Universal Robots URScript: spheremod.script

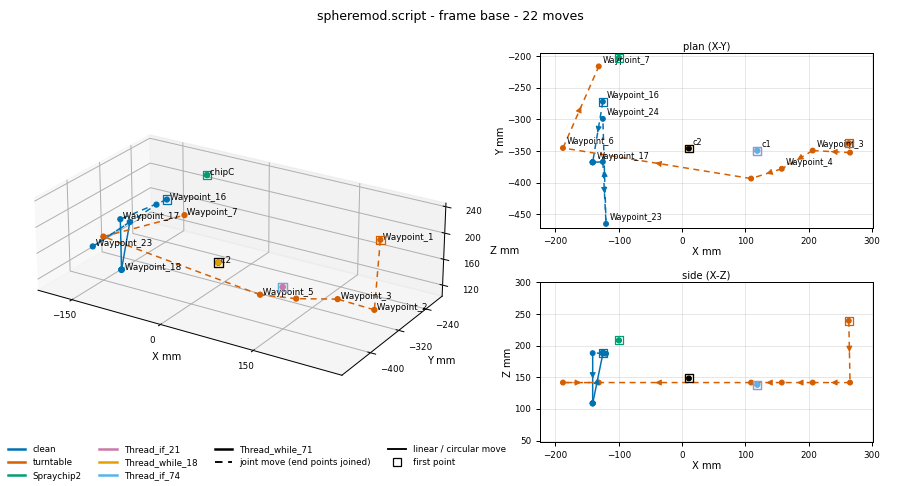
[picture p0: tool path of spheremod.script in frame base, 22 of 62 moves have a stored position in this frame; points joined in program order, loops and branches not executed]
def spheremod():
  global _hidden_verificationVariable=0
  step_count_fb48d3ff_0c9f_4d99_a765_ea41926c28d5 = 0.0
  thread Step_Counter_Thread_a9617a2c_6c0b_4ca4_aaba_c79477845290():
    while (True):
      step_count_fb48d3ff_0c9f_4d99_a765_ea41926c28d5 = step_count_fb48d3ff_0c9f_4d99_a765_ea41926c28d5 + 1.0
      sync()
    end
  end
  run Step_Counter_Thread_a9617a2c_6c0b_4ca4_aaba_c79477845290()
  set_standard_analog_input_domain(0, 1)
  set_standard_analog_input_domain(1, 1)
  set_tool_analog_input_domain(0, 1)
  set_tool_analog_input_domain(1, 1)
  set_analog_outputdomain(0, 0)
  set_analog_outputdomain(1, 0)
  set_input_actions_to_default()
  set_tool_communication(False, 115200, 0, 1, 1.5, 3.5)
  set_tool_output_mode(0)
  set_tool_digital_output_mode(0, 1)
  set_tool_digital_output_mode(1, 1)
  set_tool_voltage(0)
  set_safety_mode_transition_hardness(1)
  set_gravity([0.0, 0.0, 9.82])
  set_target_payload(0.530000, [0.009000, -0.039000, 0.092000], [0.000534, 0.000534, 0.000534, 0.000000, 0.000000, 0.000000])
  set_tcp(p[0.0,0.0,0.11,0.0,0.0,0.0])
  global Al_plate=p[0.12405209206180495,-0.2666666051843552,0.020008101224669964,-9.276623980477388E-5,1.8107917580596192E-5,3.1233857134705927]
  global Frame2x2=p[0.18266245434305164,-0.34273121659514855,0.026002571110600767,-2.225423529876215E-4,3.0110667546023537E-4,3.1233976058306383]
  global Plane_1=p[0.0,0.0,0.0,0.0,0.0,0.0]
  global URlogoTutorial=p[-0.08178353973148575,-0.3363174165299142,0.04788621506469384,-3.9746155723688456E-5,-3.4682148779121894E-5,-1.5668291789091222]
  global carousel=p[0.13865255139760183,-0.25132593351268107,0.051531504137083003,-4.453572132438073E-5,-1.3071222590669835E-4,-3.1349676625391965]
  global carouselrod=p[0.2020731702281844,-0.34951442511341274,0.1947611446273096,3.139766958234101,-0.10689428010274801,-1.1796370330365635E-5]
  global paper=p[-0.09670794781244417,-0.3283412964648025,0.027665994240809913,-3.2057893450593004E-5,2.867088716161181E-5,-1.6085327915291054]
  global rod=p[0.13368013097420872,-0.41123185103490206,0.09926814901395645,2.2214229924093103,-2.2214158162465862,-2.9165882738638143E-5]
  global timer_1=0
  global c1_p=p[.118888830935, -.349388142069, .138324188628, -3.141139658809, .028493427521, .002872972354]
  global c1_q=[-0.8784921805011194, -1.7871462307372035, -1.5894867181777954, -1.3364218038371583, 1.5709693431854248, 3.850743532180786]
  global c2_p=p[.010821857253, -.346022311091, .148298540443, -3.141186124538, .028346003463, .002753345138]
  global c2_q=[-1.1497486273394983, -1.679014345208639, -1.6702346801757812, -1.3633616727641602, 1.5705503225326538, 3.57938551902771]
  global Waypoint_16_p=p[-.125097928533, -.271984222044, .188211676824, -3.139810722578, .105446315311, .000070958927]
  global Waypoint_16_q=[-1.5480602423297327, -1.4491210740855713, -1.7099264860153198, -1.552596167927124, 1.5715936422348022, 3.23006010055542]
  global Waypoint_17_p=p[-.141183217597, -.367684006591, .188213447751, 3.139821760490, -.105397104768, -.000067867997]
  global Waypoint_17_q=[-1.597567383443014, -1.8740092716612757, -1.241610050201416, -1.5960084400572718, 1.5719740390777588, 3.1803600788116455]
  global Waypoint_18_p=p[-.141178244459, -.367687282910, .108904454765, 3.139816402425, -.105408093734, -.000060814483]
  global Waypoint_18_q=[-1.5975983778582972, -1.9245020351805628, -1.550661325454712, -1.2364590925029297, 1.5723340511322021, 3.1807193756103516]
  global Waypoint_19_p=p[-.141189357305, -.367687267469, .108915260822, 3.121780755938, .351957921543, -.000099281586]
  global Waypoint_19_q=[-1.5976179281817835, -1.9244748554625453, -1.550661325454712, -1.2364507478526612, 1.572314977645874, 2.889045000076294]
  global Waypoint_20_p=p[-.141176698746, -.367682773595, .108907204798, -3.111042719163, .436975672702, .000063164110]
  global Waypoint_20_q=[-1.5975945631610315, -1.9244939289488734, -1.5506495237350464, -1.2365017098239441, 1.5723340511322021, 3.3926987648010254]
  global Waypoint_21_p=p[-.141174078526, -.367696805030, .108909057026, 3.139786221315, -.105395786134, -.000060564502]
  global Waypoint_21_q=[-1.597586456929342, -1.9245058498778285, -1.5506460666656494, -1.2364399594119568, 1.5723340511322021, 3.1807241439819336]
  global Waypoint_22_p=p[-.125093999497, -.367099400456, .187371407622, 3.139783011421, -.105392168035, -.000053869150]
  global Waypoint_22_q=[-1.5538747946368616, -1.846323629418844, -1.2822730541229248, -1.5829936466612757, 1.5719654560089111, 3.224064588546753]
  global Waypoint_23_p=p[-.120064390322, -.465070651334, .187365924664, 2.700279766902, -.088400420341, .019763045538]
  global Waypoint_23_q=[-1.5412524382220667, -1.9475652180113734, -1.406833291053772, -0.9173591893962403, 1.5603561401367188, 3.2332537174224854]
  global Waypoint_24_p=p[-.125099110421, -.299097154487, .189878767902, 3.139750209928, -.105401717856, -.000111797080]
  global Waypoint_24_q=[-1.550074879323141, -1.5617311683348198, -1.5979981422424316, -1.5518303674510499, 1.5716702938079834, 3.2279696464538574]
  global Waypoint_1_p=p[.263501689877, -.337317763427, .239349489480, 3.139797243720, -.105347053477, -.000037720516]
  global Waypoint_1_q=[-0.5959728399859827, -2.1057659588255824, -0.6533136367797852, -1.9525557957091273, 1.5718059539794922, 4.181682586669922]
  global Waypoint_2_p=p[.265438435610, -.352444474661, .141740907029, 3.139726376264, -.105360108121, -.000022031768]
  global Waypoint_2_q=[-0.6231134573565882, -2.1016999683775843, -1.126999020576477, -1.4828875821879883, 1.5722739696502686, 4.154912948608398]
  global Waypoint_3_p=p[.206441973084, -.349241721273, .141737893294, 3.139734184252, -.105329347268, -.000022485776]
  global Waypoint_3_q=[-0.7073677221881312, -1.9410401783385218, -1.3681066036224365, -1.4024366003325959, 1.5721865892410278, 4.070710182189941]
  global Waypoint_4_p=p[.157616611756, -.378012026932, .141738203587, 3.139764187573, -.105376653239, -.000076760662]
  global Waypoint_4_q=[-0.8494070211993616, -1.9579774341978968, -1.3439116477966309, -1.409730003481247, 1.5722019672393799, 3.928692579269409]
  global Waypoint_5_p=p[.109134761588, -.393436595889, .141742225598, 3.139732501163, -.105376381431, -.000050533951]
  global Waypoint_5_q=[-0.972816292439596, -1.9523960552611292, -1.3519116640090942, -1.4072665137103577, 1.5721949338912964, 3.805286407470703]
  global Waypoint_6_p=p[-.188131250090, -.345166366147, .141750553976, 3.139727051239, -.105353578209, -.000024875816]
  global Waypoint_6_q=[-1.7293437162982386, -1.8864180050291957, -1.4439769983291626, -1.381135032778122, 1.572224736213684, 3.0487747192382812]
  global Waypoint_7_p=p[-.131564048097, -.216205376465, .141741700579, 3.139714533984, -.105382776464, -.000044168049]
  global Waypoint_7_q=[-1.572542969380514, -1.2417927545360108, -2.0833356380462646, -1.3863917154124756, 1.571577787399292, 3.2058310508728027]
  global chipC_p=p[-.099703384862, -.202952364142, .208439850600, 3.139657619359, -.105437397760, -.000145108772]
  global chipC_q=[-1.4082325140582483, -1.0998719197562714, -1.8470008373260498, -1.7646123371519984, 1.5710017681121826, 3.3699307441711426]
  global Waypoint_15_p=p[-.099704296715, -.202951379992, .208432580258, 3.139670120847, -.105426183766, -.000160358536]
  global Waypoint_15_q=[-1.4082286993609827, -1.099871740942337, -1.8470300436019897, -1.764597078362936, 1.5709946155548096, 3.369927167892456]
  global timer_1_is_counting=False
  thread Timer_Thread():
    while (True):
      if (timer_1_is_counting):
        timer_1 = timer_1 + get_steptime()
      end
      sync()
    end
  end
  run Timer_Thread()
  def CircleAllangles():
    $ 181 "CircleAllangles" "noBreak"
    $ 182 "p0≔p[c[0]+r,c[1],c[2],c[3],c[4],c[5]-1.5*A]"
    global p0=p[c[0]+r,c[1],c[2],c[3],c[4],c[5]-1.5*A]
    $ 183 "p45≔p[c[0]+0.71*r,c[1]+0.71*r,c[2],c[3]-A/1.1,c[4],c[5]-A/1.1]"
    global p45=p[c[0]+0.71*r,c[1]+0.71*r,c[2],c[3]-A/1.1,c[4],c[5]-A/1.1]
    $ 184 "p90≔p[c[0],c[1]+r,c[2],c[3]-A,c[4],c[5]]"
    global p90=p[c[0],c[1]+r,c[2],c[3]-A,c[4],c[5]]
    $ 185 "p135≔p[c[0]-0.71*r,c[1]+0.71*r,c[2],c[3]-A/1.1,c[4],c[5]+A/1.1]"
    global p135=p[c[0]-0.71*r,c[1]+0.71*r,c[2],c[3]-A/1.1,c[4],c[5]+A/1.1]
    $ 186 "p180≔p[c[0]-r,c[1],c[2],c[3],c[4],c[5]+1.5*A]"
    global p180=p[c[0]-r,c[1],c[2],c[3],c[4],c[5]+1.5*A]
    $ 187 "p225≔p[c[0]-0.71*r,c[1]-0.71*r,c[2],c[3]+A/1.1,c[4],c[5]+A/1.1]"
    global p225=p[c[0]-0.71*r,c[1]-0.71*r,c[2],c[3]+A/1.1,c[4],c[5]+A/1.1]
    $ 188 "p270≔p[c[0],c[1]-r,c[2],c[3]+A,c[4],c[5]]"
    global p270=p[c[0],c[1]-r,c[2],c[3]+A,c[4],c[5]]
    $ 189 "p315≔p[c[0]+0.71*r,c[1]-0.71*r,c[2],c[3]+A/1.1,c[4],c[5]-A/1.1]"
    global p315=p[c[0]+0.71*r,c[1]-0.71*r,c[2],c[3]+A/1.1,c[4],c[5]-A/1.1]
    $ 190 "Set atomization=On"
    set_standard_digital_out(1, True)
    $ 191 "Set triggersolenoid=On"
    set_standard_digital_out(0, True)
    $ 192 "MoveL"
    $ 193 "p0" "breakAfter"
    set_tcp(p[0.0,0.0,0.11,0.0,0.0,0.0])
    movel(p0, a=1.3, v=0.35, r=0.005)
    $ 195 "p45" "breakAfter"
    set_tcp(p[0.0,0.0,0.11,0.0,0.0,0.0])
    movel(p45, a=1.3, v=0.35, r=0.005)
    $ 197 "p90" "breakAfter"
    set_tcp(p[0.0,0.0,0.11,0.0,0.0,0.0])
    movel(p90, a=1.3, v=0.35, r=0.005)
    $ 199 "p135" "breakAfter"
    set_tcp(p[0.0,0.0,0.11,0.0,0.0,0.0])
    movel(p135, a=1.3, v=0.35, r=0.005)
    $ 201 "p180" "breakAfter"
    set_tcp(p[0.0,0.0,0.11,0.0,0.0,0.0])
    movel(p180, a=1.3, v=0.35, r=0.005)
    $ 206 "p225" "breakAfter"
    set_tcp(p[0.0,0.0,0.11,0.0,0.0,0.0])
    movel(p225, a=1.3, v=0.35, r=0.005)
    $ 208 "p270" "breakAfter"
    set_tcp(p[0.0,0.0,0.11,0.0,0.0,0.0])
    movel(p270, a=1.3, v=0.35, r=0.005)
    $ 210 "p315" "breakAfter"
    set_tcp(p[0.0,0.0,0.11,0.0,0.0,0.0])
    movel(p315, a=1.3, v=0.35, r=0.005)
    $ 212 "p0" "breakAfter"
    set_tcp(p[0.0,0.0,0.11,0.0,0.0,0.0])
    movel(p0, a=1.3, v=0.35, r=0.005)
    $ 214 "p45" "breakAfter"
    set_tcp(p[0.0,0.0,0.11,0.0,0.0,0.0])
    movel(p45, a=1.3, v=0.35, r=0.005)
    $ 219 "p90" "breakAfter"
    set_tcp(p[0.0,0.0,0.11,0.0,0.0,0.0])
    movel(p90, a=1.3, v=0.35, r=0.005)
    $ 226 "Set atomization=Off"
    set_standard_digital_out(1, False)
    $ 227 "Set triggersolenoid=Off"
    set_standard_digital_out(0, False)
  end
  def clean():
    $ 228 "clean" "noBreak"
    $ 229 "MoveJ"
    $ 230 "Waypoint_16" "breakAfter"
    movej(get_inverse_kin(Waypoint_16_p, qnear=Waypoint_16_q), a=1.3962634015954636, v=1.0471975511965976)
    $ 231 "Waypoint_17" "breakAfter"
    movej(get_inverse_kin(Waypoint_17_p, qnear=Waypoint_17_q), a=1.3962634015954636, v=1.0471975511965976)
    $ 232 "MoveL"
    $ 233 "Waypoint_18" "breakAfter"
    movel(Waypoint_18_p, a=1.2, v=0.05)
    $ 234 "MoveL"
    $ 235 "Waypoint_19" "breakAfter"
    movel(Waypoint_19_p, a=1.2, v=0.05)
    $ 236 "MoveL"
    $ 237 "Waypoint_20" "breakAfter"
    movel(Waypoint_20_p, a=1.2, v=0.05)
    $ 238 "MoveL"
    $ 239 "Waypoint_21" "breakAfter"
    movel(Waypoint_21_p, a=1.2, v=0.05)
    $ 240 "MoveL"
    $ 241 "Waypoint_22" "breakAfter"
    movel(Waypoint_22_p, a=1.2, v=0.25)
    $ 242 "MoveJ"
    $ 243 "Waypoint_23" "breakAfter"
    movej(get_inverse_kin(Waypoint_23_p, qnear=Waypoint_23_q), a=1.3962634015954636, v=1.0471975511965976)
    $ 244 "Set atomization=On"
    set_standard_digital_out(1, True)
    $ 245 "Set triggersolenoid=On"
    set_standard_digital_out(0, True)
    $ 246 "Wait: 0.2"
    sleep(0.2)
    $ 247 "Set atomization=Off"
    set_standard_digital_out(1, False)
    $ 248 "Set triggersolenoid=Off"
    set_standard_digital_out(0, False)
    $ 249 "MoveJ"
    $ 250 "Waypoint_24" "breakAfter"
    movej(get_inverse_kin(Waypoint_24_p, qnear=Waypoint_24_q), a=1.3962634015954636, v=1.0471975511965976)
  end
  def turntable():
    $ 251 "turntable" "noBreak"
    $ 252 "MoveJ"
    $ 253 "Waypoint_1" "breakAfter"
    set_tcp(p[0.0,0.0,0.11,0.0,0.0,0.0])
    movej(get_inverse_kin(pose_trans(carouselrod, pose_trans(p[-.225374943892, -.334963115589, .194760490875, -3.139766958133, .106894280099, .000011796372], Waypoint_1_p)), qnear=Waypoint_1_q), a=1.3962634015954636, v=0.5235987755982988, r=0.02)
    $ 254 "Waypoint_2" "breakAfter"
    set_tcp(p[0.0,0.0,0.11,0.0,0.0,0.0])
    movej(get_inverse_kin(pose_trans(carouselrod, pose_trans(p[-.225374943892, -.334963115589, .194760490875, -3.139766958133, .106894280099, .000011796372], Waypoint_2_p)), qnear=Waypoint_2_q), a=1.3962634015954636, v=0.5235987755982988, r=0.02)
    $ 255 "Waypoint_3" "breakAfter"
    set_tcp(p[0.0,0.0,0.11,0.0,0.0,0.0])
    movej(get_inverse_kin(pose_trans(carouselrod, pose_trans(p[-.225374943892, -.334963115589, .194760490875, -3.139766958133, .106894280099, .000011796372], Waypoint_3_p)), qnear=Waypoint_3_q), a=1.3962634015954636, v=0.5235987755982988, r=0.02)
    $ 256 "Waypoint_4" "breakAfter"
    set_tcp(p[0.0,0.0,0.11,0.0,0.0,0.0])
    movej(get_inverse_kin(pose_trans(carouselrod, pose_trans(p[-.225374943892, -.334963115589, .194760490875, -3.139766958133, .106894280099, .000011796372], Waypoint_4_p)), qnear=Waypoint_4_q), a=1.3962634015954636, v=0.5235987755982988, r=0.02)
    $ 257 "Waypoint_5" "breakAfter"
    set_tcp(p[0.0,0.0,0.11,0.0,0.0,0.0])
    movej(get_inverse_kin(pose_trans(carouselrod, pose_trans(p[-.225374943892, -.334963115589, .194760490875, -3.139766958133, .106894280099, .000011796372], Waypoint_5_p)), qnear=Waypoint_5_q), a=1.3962634015954636, v=0.5235987755982988, r=0.02)
    $ 258 "MoveJ"
    $ 259 "Waypoint_6" "breakAfter"
    movej(get_inverse_kin(pose_trans(carouselrod, pose_trans(p[-.225374943892, -.334963115589, .194760490875, -3.139766958133, .106894280099, .000011796372], Waypoint_6_p)), qnear=Waypoint_6_q), a=1.3962634015954636, v=0.3141592653589793)
    $ 260 "Wait: 1.0"
    sleep(1.0)
    $ 261 "MoveJ"
    $ 262 "Waypoint_7" "breakAfter"
    movej(get_inverse_kin(pose_trans(carouselrod, pose_trans(p[-.225374943892, -.334963115589, .194760490875, -3.139766958133, .106894280099, .000011796372], Waypoint_7_p)), qnear=Waypoint_7_q), a=1.3962634015954636, v=1.0471975511965976, r=0.02)
  end
  def Spraychip2():
    $ 263 "Spraychip2" "noBreak"
    $ 264 "MoveJ"
    $ 265 "chipC" "breakAfter"
    movej(get_inverse_kin(chipC_p, qnear=chipC_q), a=1.3962634015954636, v=1.0471975511965976)
    $ 266 "c≔chipC"
    global c=chipC_p
    $ 267 "rc≔27/1000"
    global rc=27/1000
    $ 268 "p0≔p[c[0]+rc,c[1],c[2],c[3],c[4],c[5]-1.5*0]"
    global p0=p[c[0]+rc,c[1],c[2],c[3],c[4],c[5]-1.5*0]
    $ 269 "p45≔p[c[0]+0.71*rc,c[1]+0.71*rc,c[2],c[3]-0/1.1,c[4],c[5]-0/1.1]"
    global p45=p[c[0]+0.71*rc,c[1]+0.71*rc,c[2],c[3]-0/1.1,c[4],c[5]-0/1.1]
    $ 270 "p90≔p[c[0],c[1]+rc,c[2],c[3]-0,c[4],c[5]]"
    global p90=p[c[0],c[1]+rc,c[2],c[3]-0,c[4],c[5]]
    $ 271 "p135≔p[c[0]-0.71*rc,c[1]+0.71*rc,c[2],c[3]-0/1.1,c[4],c[5]+0/1.1]"
    global p135=p[c[0]-0.71*rc,c[1]+0.71*rc,c[2],c[3]-0/1.1,c[4],c[5]+0/1.1]
    $ 272 "p180≔p[c[0]-rc,c[1],c[2],c[3],c[4],c[5]+1.5*0]"
    global p180=p[c[0]-rc,c[1],c[2],c[3],c[4],c[5]+1.5*0]
    $ 273 "p225≔p[c[0]-0.71*rc,c[1]-0.71*rc,c[2],c[3]+0/1.1,c[4],c[5]+0/1.1]"
    global p225=p[c[0]-0.71*rc,c[1]-0.71*rc,c[2],c[3]+0/1.1,c[4],c[5]+0/1.1]
    $ 274 "p270≔p[c[0],c[1]-rc,c[2],c[3]+0,c[4],c[5]]"
    global p270=p[c[0],c[1]-rc,c[2],c[3]+0,c[4],c[5]]
    $ 275 "p315≔p[c[0]+0.71*rc,c[1]-0.71*rc,c[2],c[3]+0/1.1,c[4],c[5]-0/1.1]"
    global p315=p[c[0]+0.71*rc,c[1]-0.71*rc,c[2],c[3]+0/1.1,c[4],c[5]-0/1.1]
    $ 276 "Set atomization=On"
    set_standard_digital_out(1, True)
    $ 277 "Set triggersolenoid=On"
    set_standard_digital_out(0, True)
    $ 278 "MoveL"
    $ 279 "p0" "breakAfter"
    set_tcp(p[0.0,0.0,0.11,0.0,0.0,0.0])
    movel(p0, a=1.3, v=0.085, r=0.01)
    $ 280 "p45" "breakAfter"
    set_tcp(p[0.0,0.0,0.11,0.0,0.0,0.0])
    movel(p45, a=1.3, v=0.085, r=0.01)
    $ 281 "p90" "breakAfter"
    set_tcp(p[0.0,0.0,0.11,0.0,0.0,0.0])
    movel(p90, a=1.3, v=0.085, r=0.01)
    $ 282 "p135" "breakAfter"
    set_tcp(p[0.0,0.0,0.11,0.0,0.0,0.0])
    movel(p135, a=1.3, v=0.085, r=0.01)
    $ 283 "p180" "breakAfter"
    set_tcp(p[0.0,0.0,0.11,0.0,0.0,0.0])
    movel(p180, a=1.3, v=0.085, r=0.01)
    $ 284 "Set triggersolenoid=Off"
    set_standard_digital_out(0, False)
    $ 285 "Wait: 0.1"
    sleep(0.1)
    $ 286 "Set triggersolenoid=On"
    set_standard_digital_out(0, True)
    $ 287 "p225" "breakAfter"
    set_tcp(p[0.0,0.0,0.11,0.0,0.0,0.0])
    movel(p225, a=1.3, v=0.085, r=0.01)
    $ 288 "p270" "breakAfter"
    set_tcp(p[0.0,0.0,0.11,0.0,0.0,0.0])
    movel(p270, a=1.3, v=0.085, r=0.01)
    $ 289 "p315" "breakAfter"
    set_tcp(p[0.0,0.0,0.11,0.0,0.0,0.0])
    movel(p315, a=1.3, v=0.085, r=0.01)
    $ 290 "p0" "breakAfter"
    set_tcp(p[0.0,0.0,0.11,0.0,0.0,0.0])
    movel(p0, a=1.3, v=0.085, r=0.01)
    $ 291 "p45" "breakAfter"
    set_tcp(p[0.0,0.0,0.11,0.0,0.0,0.0])
    movel(p45, a=1.3, v=0.085, r=0.01)
    $ 292 "Set triggersolenoid=Off"
    set_standard_digital_out(0, False)
    $ 293 "Wait: 0.1"
    sleep(0.1)
    $ 294 "Set triggersolenoid=On"
    set_standard_digital_out(0, True)
    $ 295 "p90" "breakAfter"
    set_tcp(p[0.0,0.0,0.11,0.0,0.0,0.0])
    movel(p90, a=1.3, v=0.085, r=0.01)
    $ 296 "p135" "breakAfter"
    set_tcp(p[0.0,0.0,0.11,0.0,0.0,0.0])
    movel(p135, a=1.3, v=0.085, r=0.01)
    $ 297 "p180" "breakAfter"
    set_tcp(p[0.0,0.0,0.11,0.0,0.0,0.0])
    movel(p180, a=1.3, v=0.085, r=0.01)
    $ 298 "p225" "breakAfter"
    set_tcp(p[0.0,0.0,0.11,0.0,0.0,0.0])
    movel(p225, a=1.3, v=0.085, r=0.01)
    $ 299 "p270" "breakAfter"
    set_tcp(p[0.0,0.0,0.11,0.0,0.0,0.0])
    movel(p270, a=1.3, v=0.085, r=0.01)
    $ 300 "p315" "breakAfter"
    set_tcp(p[0.0,0.0,0.11,0.0,0.0,0.0])
    movel(p315, a=1.3, v=0.085, r=0.01)
    $ 301 "p0" "breakAfter"
    set_tcp(p[0.0,0.0,0.11,0.0,0.0,0.0])
    movel(p0, a=1.3, v=0.085, r=0.01)
    $ 302 "MoveJ"
    $ 303 "Waypoint_15" "breakAfter"
    movej(get_inverse_kin(Waypoint_15_p, qnear=Waypoint_15_q), a=1.3962634015954636, v=1.0471975511965976)
    $ 304 "Wait: 0.2"
    sleep(0.2)
    $ 305 "Set atomization=Off"
    set_standard_digital_out(1, False)
    $ 306 "Set triggersolenoid=Off"
    set_standard_digital_out(0, False)
  end
  while (True):
    $ 2 "Robot Program"
    $ 3 "'Program to be used for part #124517-035 sphere mod'"
    # 'Program to be used for part #124517-035 sphere mod'
    $ 4 "'Program rev ___: mm/dd/yy note'"
    # 'Program rev ___: mm/dd/yy note'
    $ 5 "timer_1: Start"
    timer_1_is_counting = True
    $ 6 "r≔1/1000"
    global r=1/1000
    $ 7 "A≔3*3.1416/180"
    global A=3*3.1416/180
    $ 8 "Loop_1≔1"
    global Loop_1=1
    $ 10 "partnum≔2"
    global partnum=2
    $ 12 "coatnum≔2"
    global coatnum=2
    $ 13 "sidenum≔2"
    global sidenum=2
    $ 14 "If partnum≤sidenum"
    global thread_flag_14=0
    thread Thread_if_14():
      $ 15 "Loop (coatnum)>0"
      thread Thread_while_15():
        while (True):
          $ 16 "partleft≔partnum"
          global partleft=partnum
          $ 17 "loopnum≔1"
          global loopnum=1
          $ 18 "Loop partleft>0"
          thread Thread_while_18():
            while (True):
              $ 19 "Call clean"
              clean()
              $ 20 "Call Spraychip2"
              Spraychip2()
              $ 21 "If loopnum≟1 or loopnum≟3 or loopnum≟5 or loopnum≟7 or loopnum≟9 or loopnum≟11"
              global thread_flag_21=0
              thread Thread_if_21():
                $ 22 "MoveJ"
                $ 23 "c1" "breakAfter"
                movej(get_inverse_kin(c1_p, qnear=c1_q), a=1.3962634015954636, v=1.0471975511965976)
                $ 24 "c≔c1"
                global c=c1_p
                $ 25 "Call CircleAllangles"
                CircleAllangles()
                $ 26 "x2≔p[c[0]-0.048,c[1],c[2],c[3],c[4],c[5]]"
                global x2=p[c[0]-0.048,c[1],c[2],c[3],c[4],c[5]]
                $ 27 "x3≔p[c[0]-0.048,c[1]+0.048,c[2],c[3],c[4],c[5]]"
                global x3=p[c[0]-0.048,c[1]+0.048,c[2],c[3],c[4],c[5]]
                $ 28 "x4≔p[c[0],c[1]+0.048,c[2],c[3],c[4],c[5]]"
                global x4=p[c[0],c[1]+0.048,c[2],c[3],c[4],c[5]]
                $ 29 "MoveJ"
                $ 30 "x2" "breakAfter"
                movej(x2, a=1.3962634015954636, v=1.0471975511965976)
                $ 31 "c≔x2"
                global c=x2
                $ 32 "Call CircleAllangles"
                CircleAllangles()
                $ 33 "MoveJ"
                $ 34 "x3" "breakAfter"
                movej(x3, a=1.3962634015954636, v=1.0471975511965976)
                $ 35 "c≔x3"
                global c=x3
                $ 36 "Call CircleAllangles"
                CircleAllangles()
                $ 37 "MoveJ"
                $ 38 "x4" "breakAfter"
                movej(x4, a=1.3962634015954636, v=1.0471975511965976)
                $ 39 "c≔x4"
                global c=x4
                $ 40 "Call CircleAllangles"
                CircleAllangles()
                thread_flag_21 = 1
              end
              if (loopnum == 1  or  loopnum == 3  or  loopnum == 5  or  loopnum == 7  or  loopnum == 9  or  loopnum == 11):
                global thread_handler_21=run Thread_if_21()
                while (thread_flag_21 == 0):
                  if not(loopnum == 1  or  loopnum == 3  or  loopnum == 5  or  loopnum == 7  or  loopnum == 9  or  loopnum == 11):
                    kill thread_handler_21
                    thread_flag_21 = 2
                  else:
                    sync()
                  end
                end
              else:
                thread_flag_21 = 2
              end
              if (thread_flag_21 == 2):
                $ 41 "Else" "noBreak"
                $ 42 "MoveJ"
                $ 43 "c2" "breakAfter"
                movej(get_inverse_kin(c2_p, qnear=c2_q), a=1.3962634015954636, v=1.0471975511965976)
                $ 44 "c≔c2"
                global c=c2_p
                $ 45 "Call CircleAllangles"
                CircleAllangles()
                $ 46 "x2≔p[c[0]-0.048,c[1],c[2],c[3],c[4],c[5]]"
                global x2=p[c[0]-0.048,c[1],c[2],c[3],c[4],c[5]]
                $ 47 "x3≔p[c[0]-0.048,c[1]+0.048,c[2],c[3],c[4],c[5]]"
                global x3=p[c[0]-0.048,c[1]+0.048,c[2],c[3],c[4],c[5]]
                $ 48 "x4≔p[c[0],c[1]+0.048,c[2],c[3],c[4],c[5]]"
                global x4=p[c[0],c[1]+0.048,c[2],c[3],c[4],c[5]]
                $ 49 "MoveJ"
                $ 50 "x2" "breakAfter"
                movej(x2, a=1.3962634015954636, v=1.0471975511965976)
                $ 51 "c≔x2"
                global c=x2
                $ 52 "Call CircleAllangles"
                CircleAllangles()
                $ 53 "MoveJ"
                $ 54 "x3" "breakAfter"
                movej(x3, a=1.3962634015954636, v=1.0471975511965976)
                $ 55 "c≔x3"
                global c=x3
                $ 56 "Call CircleAllangles"
                CircleAllangles()
                $ 57 "MoveJ"
                $ 58 "x4" "breakAfter"
                movej(x4, a=1.3962634015954636, v=1.0471975511965976)
                $ 59 "c≔x4"
                global c=x4
                $ 60 "Call CircleAllangles"
                CircleAllangles()
              end
              $ 61 "loopnum≔loopnum+1"
              global loopnum=loopnum+1
              $ 62 "partleft≔partleft-1"
              global partleft=partleft-1
            end
          end
          if (partleft>0):
            global thread_handler_18=run Thread_while_18()
            while (partleft>0):
              sync()
            end
            kill thread_handler_18
          end
          $ 63 "i≔0"
          global i=0
          $ 64 "coatnum≔coatnum-1"
          global coatnum=coatnum-1
        end
      end
      if ((coatnum)>0):
        global thread_handler_15=run Thread_while_15()
        while ((coatnum)>0):
          sync()
        end
        kill thread_handler_15
      end
      $ 65 "Halt"
      halt
      thread_flag_14 = 1
    end
    if (partnum <= sidenum):
      global thread_handler_14=run Thread_if_14()
      while (thread_flag_14 == 0):
        if not(partnum <= sidenum):
          kill thread_handler_14
          thread_flag_14 = 2
        else:
          sync()
        end
      end
    else:
      thread_flag_14 = 2
    end
    if (thread_flag_14 == 2):
      $ 66 "Else" "noBreak"
      $ 67 "Loop (coatnum)>0"
      thread Thread_while_67():
        while (True):
          $ 68 "partleft≔partnum"
          global partleft=partnum
          $ 69 "loopnum≔1"
          global loopnum=1
          $ 70 "turnnum≔0"
          global turnnum=0
          $ 71 "Loop partleft>0"
          thread Thread_while_71():
            while (True):
              $ 72 "Call clean"
              clean()
              $ 73 "Call Spraychip2"
              Spraychip2()
              $ 74 "If loopnum≟1 or loopnum≟3 or loopnum≟5 or loopnum≟7 or loopnum≟9 or loopnum≟11"
              global thread_flag_74=0
              thread Thread_if_74():
                $ 104 "MoveJ"
                $ 105 "c1" "breakAfter"
                movej(get_inverse_kin(c1_p, qnear=c1_q), a=1.3962634015954636, v=1.0471975511965976)
                $ 106 "c≔c1"
                global c=c1_p
                $ 107 "Call CircleAllangles"
                CircleAllangles()
                $ 108 "x2≔p[c[0]-0.048,c[1],c[2],c[3],c[4],c[5]]"
                global x2=p[c[0]-0.048,c[1],c[2],c[3],c[4],c[5]]
                $ 109 "x3≔p[c[0]-0.048,c[1]+0.048,c[2],c[3],c[4],c[5]]"
                global x3=p[c[0]-0.048,c[1]+0.048,c[2],c[3],c[4],c[5]]
                $ 110 "x4≔p[c[0],c[1]+0.048,c[2],c[3],c[4],c[5]]"
                global x4=p[c[0],c[1]+0.048,c[2],c[3],c[4],c[5]]
                $ 111 "MoveJ"
                $ 112 "x2" "breakAfter"
                movej(x2, a=1.3962634015954636, v=1.0471975511965976)
                $ 113 "c≔x2"
                global c=x2
                $ 114 "Call CircleAllangles"
                CircleAllangles()
                $ 115 "MoveJ"
                $ 116 "x3" "breakAfter"
                movej(x3, a=1.3962634015954636, v=1.0471975511965976)
                $ 117 "c≔x3"
                global c=x3
                $ 118 "Call CircleAllangles"
                CircleAllangles()
                $ 119 "MoveJ"
                $ 120 "x4" "breakAfter"
                movej(x4, a=1.3962634015954636, v=1.0471975511965976)
                $ 121 "c≔x4"
                global c=x4
                $ 122 "Call CircleAllangles"
                CircleAllangles()
                thread_flag_74 = 1
              end
              if (loopnum == 1  or  loopnum == 3  or  loopnum == 5  or  loopnum == 7  or  loopnum == 9  or  loopnum == 11):
                global thread_handler_74=run Thread_if_74()
                while (thread_flag_74 == 0):
                  if not(loopnum == 1  or  loopnum == 3  or  loopnum == 5  or  loopnum == 7  or  loopnum == 9  or  loopnum == 11):
                    kill thread_handler_74
                    thread_flag_74 = 2
                  else:
                    sync()
                  end
                end
              else:
                thread_flag_74 = 2
              end
              if (thread_flag_74 == 2):
                $ 123 "Else" "noBreak"
                $ 154 "MoveJ"
                $ 155 "c2" "breakAfter"
                movej(get_inverse_kin(c2_p, qnear=c2_q), a=1.3962634015954636, v=1.0471975511965976)
                $ 156 "c≔c2"
                global c=c2_p
                $ 157 "Call CircleAllangles"
                CircleAllangles()
                $ 158 "x2≔p[c[0]-0.048,c[1],c[2],c[3],c[4],c[5]]"
                global x2=p[c[0]-0.048,c[1],c[2],c[3],c[4],c[5]]
                $ 159 "x3≔p[c[0]-0.048,c[1]+0.048,c[2],c[3],c[4],c[5]]"
                global x3=p[c[0]-0.048,c[1]+0.048,c[2],c[3],c[4],c[5]]
                $ 160 "x4≔p[c[0],c[1]+0.048,c[2],c[3],c[4],c[5]]"
                global x4=p[c[0],c[1]+0.048,c[2],c[3],c[4],c[5]]
                $ 161 "MoveJ"
                $ 162 "x2" "breakAfter"
                movej(x2, a=1.3962634015954636, v=1.0471975511965976)
                $ 163 "c≔x2"
                global c=x2
                $ 164 "Call CircleAllangles"
                CircleAllangles()
                $ 165 "MoveJ"
                $ 166 "x3" "breakAfter"
                movej(x3, a=1.3962634015954636, v=1.0471975511965976)
                $ 167 "c≔x3"
                global c=x3
                $ 168 "Call CircleAllangles"
                CircleAllangles()
                $ 169 "MoveJ"
                $ 170 "x4" "breakAfter"
                movej(x4, a=1.3962634015954636, v=1.0471975511965976)
                $ 171 "c≔x4"
                global c=x4
                $ 172 "Call CircleAllangles"
                CircleAllangles()
              end
              $ 173 "loopnum≔loopnum+1"
              global loopnum=loopnum+1
              $ 174 "partleft≔partleft-1"
              global partleft=partleft-1
            end
          end
          if (partleft>0):
            global thread_handler_71=run Thread_while_71()
            while (partleft>0):
              sync()
            end
            kill thread_handler_71
          end
          $ 175 "i≔0"
          global i=0
          $ 176 "Loop (6-turnnum)>0"
          thread Thread_while_176():
            while (True):
              $ 177 "Call turntable"
              turntable()
              $ 178 "turnnum≔turnnum+1"
              global turnnum=turnnum+1
            end
          end
          if ((6-turnnum)>0):
            global thread_handler_176=run Thread_while_176()
            while ((6-turnnum)>0):
              sync()
            end
            kill thread_handler_176
          end
          $ 179 "coatnum≔coatnum-1"
          global coatnum=coatnum-1
        end
      end
      if ((coatnum)>0):
        global thread_handler_67=run Thread_while_67()
        while ((coatnum)>0):
          sync()
        end
        kill thread_handler_67
      end
      $ 180 "Halt"
      halt
    end
  end
end
